{region '#Template'}
	{attribute 'Version' := '5.0.0.0'}
	{attribute 'Tags' := '"LCID": "1031", "Text": "Universal, Object, AV"'}
	{attribute 'Tags' := '"LCID": "1033", "Text": "Universal, Object, AV"'}
	{attribute 'Using' := '"Type": "Template", "URI": "EC_ID"'}
	{attribute 'Using' := '"Type": "Template", "URI": "BA2_Param"'}
	{attribute 'Description' := '"LCID": "1031", "Text": "AV Sollwert"'}
	{attribute 'Description' := '"LCID": "1033", "Text": "AV Setpoint"'}
{endregion}
FUNCTION_BLOCK FB_BA_AV_Op_SP EXTENDS FB_BA_View
VAR_OUTPUT
	fPresentValue				: REAL;
END_VAR
VAR_INPUT CONSTANT
	SP							: FB_BA_AV_Op;		
END_VAR
VAR
END_VAR

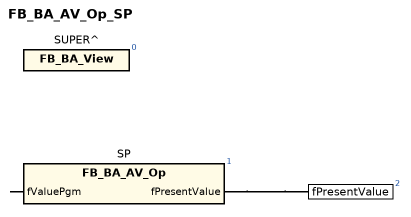
SUPER^(); // FB_BA_View
SP(); // FB_BA_AV_Op
fPresentValue := SP.fPresentValue;

METHOD FB_init : BOOL
VAR_INPUT
	bInitRetains : BOOL; // if TRUE, the retain variables are initialized (warm start / cold start)
	bInCopyCode : BOOL;  // if TRUE, the instance afterwards gets moved into the copy code (online change)
END_VAR
SP.iParent					:= THIS^;
SP.iLabel					:= LblFun_Setpoint; 
SP.eUnit					:= E_BA_Unit.eTemperature_DegreesCelsius;  
SP.fCOVIncrement			:= BA2_Param.fDefCOVIncrement;
END_METHOD

END_FUNCTION_BLOCK

(* stored: Version 1.1.0.1, ProductVersion 3.1.4024.12
   POU FB_BA_AV_Op_SP: Id {b03ca2c1-14b6-4cb7-bc1b-199f320dea5f}, SpecialFunc None
   Method FB_init: Id {5920401c-4f9a-48a9-8521-54f714708fa2} *)
